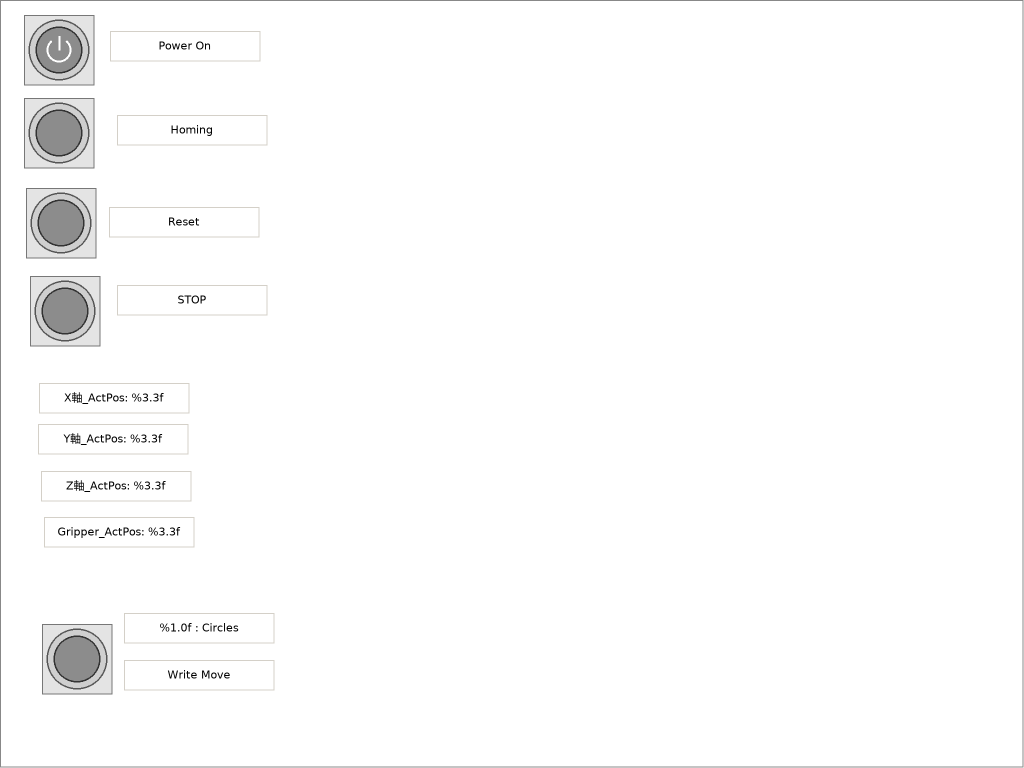
VISUALIZATION Visualization  // 1024x768
    PowerSwitch (24,15 70x70), variable: GVL.bPower, behaviour: TOGGLE, style: Switch-PowerSwitch-Gray
    PushSwitch (24,98 70x70), variable: GVL.bHome, behaviour: TAP, style: Switch-PushSwitch-Gray
    Textfield (39,383 150x30), "X軸_ActPos: %3.3f", text variable: P_WriteMotion.GVL.stAxis[E_Axis.X_Axis].NcToPlc.ActPos
    Textfield (41,471 150x30), "Z軸_ActPos: %3.3f", text variable: P_WriteMotion.GVL.stAxis[E_Axis.Z_Axis].NcToPlc.ActPos
    Textfield (38,424 150x30), "Y軸_ActPos: %3.3f", text variable: P_WriteMotion.GVL.stAxis[E_Axis.Y_Axis].NcToPlc.ActPos
    Textfield (110,31 150x30), "Power On"
    Textfield (117,115 150x30), "Homing"
    PushSwitch (26,188 70x70), variable: GVL.bReset, behaviour: TAP, style: Switch-PushSwitch-Gray
    Textfield (109,207 150x30), "Reset"
    PushSwitch (42,624 70x70), variable: GVL.bMove, behaviour: TAP, style: Switch-PushSwitch-Gray
    Textfield (124,660 150x30), "Write Move"
    PushSwitch (30,276 70x70), variable: GVL.bStop, behaviour: TAP, style: Switch-PushSwitch-Gray
    Textfield (117,285 150x30), "STOP"
    Textfield (44,517 150x30), "Gripper_ActPos: %3.3f", text variable: P_WriteMotion.GVL.stAxis[E_Axis.Gripper].NcToPlc.ActPos
    Textfield (124,613 150x30), "%1.0f : Circles", text variable: P_Circle.iEndNumberCircle
        OnMouseDown: write P_Circle.iEndNumberCircle via Default, min 1
END_VISUALIZATION

(* stored: Version 1.1.0.1, ProductVersion 3.1.4024.12
   Visu Visualization: Id {7f9da9a7-8da1-406e-844a-298ecf405691} *)
